{attribute 'qualified_only'}
{attribute 'strict'}
TYPE E_DiverterState :
(
    IDLE      := 0,
    LIFTING   := 10,
    DIVERTING := 20,
    LOWERING  := 30,
	DONE := 40,
    FAULT     := 99
);
END_TYPE

(* stored: Version 1.1.0.1, ProductVersion 3.1.4024.16
   DUT E_DiverterState: Id {b1c2d3e4-f5a6-7890-bcde-f12345678901} *)
